INTERFACE I_LowerAuthority

PROPERTY bLowerAuthorityVetoed : BOOL
GET
END_GET
SET
END_SET
END_PROPERTY

// <Arbiter Internal>
// Elevates the arbitrated BP set to something above.
// Could be another arbiter, or a BP requester/ IO, 
// or an FB that locks in a specific portion of the BP set.
METHOD ElevateRequest : BOOL 
VAR_INPUT
    HigherAuthority : I_HigherAuthority;
END_VAR
END_METHOD

PROPERTY nLowerAuthorityID : DWORD
GET
END_GET
END_PROPERTY

END_INTERFACE

(* stored: Version 1.1.0.1, ProductVersion 3.1.4022.18
   Itf I_LowerAuthority: Id {99891ecc-c797-4643-bae6-a2321f534778}
   Property bLowerAuthorityVetoed: Id {cd524703-a063-44f0-9757-e03b78361a4a}
   Get Get: Id {c3203e12-04a2-494d-b51d-7902dc37d9ee}
   Set Set: Id {ab1c501b-3928-44aa-ad03-72fc19cff2ce}
   Method ElevateRequest: Id {7b91e0f7-0ecb-4354-af40-944e958abd7b}
   Property nLowerAuthorityID: Id {aa311dee-db63-431d-b060-55dc42f449e4}
   Get Get: Id {a80bf1a7-cb9d-4dfb-870e-2eaf0155bc28} *)
